// TwinCAT 3 PLC project MAS418_PLC
// ProgramVersion: 3.1.4024.0
// libraries:
//   Tc2_Standard, * (Beckhoff Automation GmbH)
//   Tc2_System, * (Beckhoff Automation GmbH)
//   Tc3_Module, * (Beckhoff Automation GmbH)
// project tree:
//   DUTs/ Sensor_brands.TcDUT
//   GVLs/ GVL.TcGVL
//   / PlcTask.TcTTO
//   POUs/ MAIN.TcPOU, P1.TcPOU
//   Task 2/ fDegToRad.TcPOU, GVL_task2.TcGVL, P_Task2.TcPOU, ST_Timer.TcDUT, ST_Timer2.TcDUT
//   Task3/ fUpdateparam2.TcPOU, GVL_Task3.TcGVL, fUpdateparam.TcPOU, ST_Motorparam.TcDUT, P_Task3.TcPOU
// real-time tasks:
//   TASK PlcTask: cycle T#10ms, priority 20, ADS port 350

CONFIGURATION MAS418_PLC
    RESOURCE PLC ON TwinCAT3
        TASK PlcTask(INTERVAL := T#10ms, PRIORITY := 20);
        PROGRAM MAIN WITH PlcTask : MAIN;
        PROGRAM P1 WITH PlcTask : P1;
        PROGRAM P_Task2 WITH PlcTask : P_Task2;
        PROGRAM P_Task3 WITH PlcTask : P_Task3;
    END_RESOURCE
END_CONFIGURATION

// ---- DUTs/Sensor_brands.TcDUT
{attribute 'qualified_only'}
{attribute 'strict'}
TYPE Sensor_brands:
(
	Sick,
	PilZ,
	Parker:=3,
	Bosch 
)SINT;
END_TYPE

// ---- Task 2/ST_Timer.TcDUT
TYPE ST_Timer :
STRUCT
	bTimerStart   : BOOL 	   := 0;
	fbTON2 		  : TON;
	bQStatus	  : BOOL;
	tElapsedTime  : TIME	   :=T#0S;
END_STRUCT
END_TYPE

// ---- Task 2/ST_Timer2.TcDUT
TYPE ST_Timer2 :
STRUCT
	bTimerStart2	: BOOL;
	tTimer2			: TIME;
	bQStatus2	  	: BOOL;
	tElapsedTime2	: TIME;
END_STRUCT
END_TYPE

// ---- Task3/ST_Motorparam.TcDUT
TYPE ST_Motorparam :
STRUCT
	rMaxSpeed		:REAL		:= 2000;//rpm
	rMinSpeed		:REAL		:= 0;	//rpm
END_STRUCT
END_TYPE

// ---- GVLs/GVL.TcGVL
{attribute 'qualified_only'}
VAR_GLOBAL
	dtDateTime : DATE_AND_TIME := DT#2024-02-26-13:44:19;
	tTime 	   : TIME 		   := T#5S;
	aArrayTest : ARRAY[1..4] OF DATE := [D#2023-02-07, D#2023-02-08, D#2023-02-09, D#2023-02-10];
	sensor1		  : Sensor_brands;
	bTimerStart   : BOOL 	   := 0;
	tTimer 		  : TIME 	   :=T#10S;
	bQStatus	  : BOOL;
	tElapsedTime  : TIME	   :=T#0S;
END_VAR

// ---- Task 2/GVL_task2.TcGVL
{attribute 'qualified_only'}
VAR_GLOBAL
	stTimer			: ST_Timer2;
	stTimer2		: ST_Timer2:=(tTimer2:=T#5S);
	rMotor1Pos		: REAL;
END_VAR

// ---- Task3/GVL_Task3.TcGVL
{attribute 'qualified_only'}
VAR_GLOBAL
	stMotorParam1		: ST_Motorparam;
	stMotorParam2		: ST_Motorparam;
END_VAR

// ---- POUs/MAIN.TcPOU
PROGRAM MAIN
VAR
END_VAR

P1();
P_Task2();

END_PROGRAM

// ---- POUs/P1.TcPOU
PROGRAM P1
VAR
	pPointer 	  : POINTER TO DATE_AND_TIME := ADR(GVL.dtDateTime);
	rRefrencetest : REFERENCE TO TIME REF=GVL.tTime;
	pArrayref 	  : REFERENCE TO ARRAY[1..4] OF DATE REF=GVL.aArrayTest;
	fbTON		  : TON;
END_VAR

pPointer^ := DT#2023-02-08-15:31:19;

rRefrencetest := T#1S;

pArrayref[3] :=D#2023-02-25;

GVL.sensor1 := Sensor_brands.Parker;

fbTON (IN:=GVL.bTimerStart, PT:= GVL.tTimer, Q=>GVL.bQStatus, ET=>GVL.tElapsedTime);

END_PROGRAM

// ---- Task 2/P_Task2.TcPOU
PROGRAM P_Task2
VAR
	fbTOF		: TOF;
	functest	:REAL;
	degval 		:REAL:=180;
END_VAR

fbTOF(
	IN		:=GVL_task2.stTimer2.bTimerStart2,
	PT		:=GVL_task2.stTimer2.tTimer2,
	Q		=>GVL_task2.stTimer2.bQStatus2,
	ET		=>GVL_task2.stTimer2.tElapsedTime2
);

GVL_task2.rMotor1Pos:=fDegToRad(rDegrees:=degval);

END_PROGRAM

// ---- Task 2/fDegToRad.TcPOU
FUNCTION fDegToRad : REAL
VAR_INPUT
	rDegrees		:REAL;
END_VAR
VAR
END_VAR

fDegToRad:=((rDegrees*PI)/180);

END_FUNCTION

// ---- Task3/P_Task3.TcPOU
PROGRAM P_Task3
VAR
	fbRTrig			: R_TRIG;
	bSpeedCTRL		: BOOL;
	fSpeedValue		: REAL;
	bSpeedUpdate	: BOOL;
	x				: INT :=3;
END_VAR

fbRTrig(CLK:=bSpeedCTRL,
		Q=>bSpeedUpdate);
		
CASE x OF//Change input Motorspeed value
	1:
	 	GVL_Task3.stMotorParam1.rMaxSpeed := 1000;
	2:
	    GVL_Task3.stMotorParam1.rMaxSpeed := 2000;
	3:
		GVL_Task3.stMotorParam1.rMaxSpeed := 3000;
	4: 
		GVL_Task3.stMotorParam1.rMaxSpeed := 4000;	
END_CASE

fUpdateparam(bUpdateValue:=bSpeedUpdate,
			 fNewValue:=fSpeedValue,
			 stMotorParameters := GVL_Task3.stMotorParam1);

fUpdateparam2(bUpdateValue:=bSpeedUpdate,
			 fNewValue:=fSpeedValue,
			 stMotorParameters := GVL_Task3.stMotorParam1);

END_PROGRAM

// ---- Task3/fUpdateparam.TcPOU
FUNCTION fUpdateparam : REAL
VAR_INPUT
	bUpdateValue		: BOOL;
	fNewValue			: REAL;
	stMotorParameters	: ST_Motorparam;
	
END_VAR
VAR
END_VAR

IF bUpdateValue = TRUE THEN
	stMotorParameters.rMaxSpeed := fNewValue;
ELSE
	stMotorParameters.rMaxSpeed := stMotorParameters.rMaxSpeed;
END_IF

END_FUNCTION

// ---- Task3/fUpdateparam2.TcPOU
FUNCTION fUpdateparam2 : REAL
VAR_INPUT
	bUpdateValue		: BOOL;
	fNewValue			: REAL;
	stMotorParameters	: REFERENCE TO ST_Motorparam;
	
END_VAR
VAR
END_VAR

IF bUpdateValue = TRUE THEN
	stMotorParameters.rMaxSpeed := fNewValue;
ELSE
	stMotorParameters.rMaxSpeed := stMotorParameters.rMaxSpeed;
END_IF

END_FUNCTION
